// Mitsubishi GX Works2 project: PLC_250924최종   PLC: Q03UDE

// global labels: Global1
VAR_GLOBAL
  H속도변경 AT D10 : INT;
  H축1현재위치 AT D100 : DINT;
  H축2현재위치 AT D104 : DINT;
  H축1에러번호 AT D110 : INT;
  H축2에러번호 AT D111 : INT;
  H축1경고번호 AT D112 : INT;
  H축2경고번호 AT D113 : INT;
  H축1위치1 AT D120 : DINT;
  H축2위치2 AT D140 : DINT;
  H조그속도값 AT D160 : INT;
  H축1기동번호 AT D200 : DINT;
  축2기동 AT M1 : BOOL;
  H시작 AT M10 : BOOL;
  H속도변경버튼 AT M13 : BOOL;
  H축1위치1입력 AT M101 : BOOL;
  H축1위치2입력 AT M102 : BOOL;
  H축1위치3입력 AT M103 : BOOL;
  H축2위치1입력 AT M105 : BOOL;
  H축2위치2입력 AT M106 : BOOL;
  H축1위치1기동명령 AT M111 : BOOL;
  H축1위치2기동명령 AT M112 : BOOL;
  H축1위치3기동명령 AT M113 : BOOL;
  H축2위치1기동명령 AT M115 : BOOL;
  H축2위치2기동명령 AT M116 : BOOL;
  H조그상 AT M121 : BOOL;
  H조그하 AT M122 : BOOL;
  H조그좌 AT M123 : BOOL;
  H조그우 AT M124 : BOOL;
  H축1원점복귀 AT M125 : BOOL;
  H축2원점복귀 AT M126 : BOOL;
  H롬저장 AT M128 : BOOL;
  H축1서보정지 AT M129 : BOOL;
  H축2서보정지 AT M130 : BOOL;
  H축1기동스위치 AT M200 : BOOL;
  H축2기동스위치 AT M201 : BOOL;
  축1서보기동번호 AT U4\G1500 : INT;
  축2서보기동번호 AT U4\G1600 : INT;
  축1서보에러리셋 AT U4\G1502 : INT;
  축2서보에러리셋 AT U4\G1602 : INT;
  축1조그스피드값 AT U4\G1518 : DINT;
  축2조그스피드값 AT U4\G1618 : DINT;
  서보롬쓰기 AT U4\G1900 : INT;
  축2서보현재위치 AT U4\G900 : DINT;
  축1서보이송속도 AT U4\G804 : DINT;
  축2서보이송속도 AT U4\G904 : DINT;
  축1서보에러번호 AT U4\G806 : INT;
  H축1위치2 AT D124 : DINT;
  H축1위치3 AT D128 : DINT;
  H정지 AT M11 : BOOL;
  H일시정지 AT M12 : BOOL;
  축2서보에러번호 AT U4\G906 : INT;
  축1서보경고번호 AT U4\G807 : INT;
  축2서보경고번호 AT U4\G907 : INT;
  축1원점복귀완료 AT U4\G817.4 : BOOL;
  축2원점복귀완료 AT U4\G917.4 : BOOL;
  QD75레디 AT X40 : BOOL;
  축1서보비지 AT X4C : BOOL;
  축2서보비지 AT X4D : BOOL;
  축1서보완료 AT X54 : BOOL;
  축2서보완료 AT X55 : BOOL;
  PLC레디 AT Y40 : BOOL;
  축1서보정지 AT Y44 : BOOL;
  축2서보정지 AT Y45 : BOOL;
  축1조그정기동 AT Y48 : BOOL;
  축1조그역기동 AT Y49 : BOOL;
  H축2위치1 AT D136 : DINT;
  축2조그정기동 AT Y4A : BOOL;
  H축2기동번호 AT D204 : DINT;
  축2조그역기동 AT Y4B : BOOL;
  축1서보기동 AT Y50 : BOOL;
  축2서보기동 AT Y51 : BOOL;
END_VAR
VAR_GLOBAL CONSTANT
  기계원점복귀 : INT := K9001;
END_VAR
VAR_GLOBAL
  축1서보현재위치 AT U4\G800 : DINT;
  축1기동 AT M0 : BOOL;
  in색판별완료 AT M601 : BOOL;
  in두봇완료 AT M602 : BOOL;
  in흰색게이트오픈 AT M603 : BOOL;
  in검은색게이트오픈 AT M604 : BOOL;
  in흰박스full AT M605 : BOOL;
  in검은박스full AT M606 : BOOL;
  in흰박스AMR적재완 AT M607 : BOOL;
  in검은박스AMR적재완 AT M608 : BOOL;
  out공정시작 AT M700 : BOOL;
  out색판정위치도착 AT M701 : BOOL;
  out바퀴분류위치도착 AT M702 : BOOL;
  out흰박스준비완 AT M703 : BOOL;
  out검은박스준비완 AT M704 : BOOL;
  out서보흰컨베이어도착 AT M705 : BOOL;
  out서보검은컨베이어도착 AT M706 : BOOL;
  out흰박스AMR안착 AT M707 : BOOL;
  out검은박스AMR안착 AT M708 : BOOL;
  바퀴매거진센서 AT X0 : BOOL;
  바퀴공급전진센서 AT X1 : BOOL;
  바퀴공급후진센서 AT X2 : BOOL;
  바퀴차단전진센서 AT X3 : BOOL;
  바퀴차단후진센서 AT X4 : BOOL;
  바퀴판정위치센서 AT X5 : BOOL;
  바퀴분류위치센서 AT X6 : BOOL;
  흰박스매거진센서 AT X9 : BOOL;
  흰박스공급후진센서 AT X0A : BOOL;
  흰박스공급전진센서 AT X0B : BOOL;
  흰박스차단위치센서 AT X0C : BOOL;
  흰박스도착위치센서 AT X0D : BOOL;
  검은박스매거진센서 AT X0E : BOOL;
  검은박스공급전진센서 AT X0F : BOOL;
  검은박스공급후진센서 AT X10 : BOOL;
  검은박스차단위치센서 AT X11 : BOOL;
  검은박스도착위치센서 AT X12 : BOOL;
  그리퍼전진센서 AT X15 : BOOL;
  그리퍼후진센서 AT X16 : BOOL;
  그리퍼CW센서 AT X13 : BOOL;
  그리퍼CCW센서 AT X14 : BOOL;
  H축2위치3 AT D144 : DINT;
  H축2위치3입력 AT M107 : BOOL;
  H축2위치3기동명령 AT M117 : BOOL;
  H축2위치4 AT D148 : DINT;
  H축1위치4 AT D132 : DINT;
  H축1위치4입력 AT M104 : BOOL;
  H축2위치4입력 AT M108 : BOOL;
  H축1위치4기동명령 AT M114 : BOOL;
  H축2위치4기동명령 AT M118 : BOOL;
  H에러리셋 AT M127 : BOOL;
  H축2위치5 AT D152 : DINT;
  H축2위치5입력 AT M109 : BOOL;
  H축2위치5기동명령 AT M119 : BOOL;
  비상정지버튼 AT X17 : BOOL;
  바퀴공급전진솔 AT Y20 : BOOL;
  바퀴공급후진솔 AT Y21 : BOOL;
  바퀴차단전진솔 AT Y22 : BOOL;
  바퀴차단후진솔 AT Y23 : BOOL;
  바퀴컨베이어모터구동 AT Y24 : BOOL;
  흰박스공급전진솔 AT Y25 : BOOL;
  흰박스공급후진솔 AT Y26 : BOOL;
  흰박스컨베이어모터구동 AT Y27 : BOOL;
  검은박스공급전진솔 AT Y28 : BOOL;
  검은박스공급후진솔 AT Y29 : BOOL;
  검은박스컨베이어모터구동 AT Y2A : BOOL;
  그리퍼전진솔 AT Y2B : BOOL;
  그리퍼후진솔 AT Y2C : BOOL;
  그리퍼CW솔 AT Y2D : BOOL;
  그리퍼CCW솔 AT Y2E : BOOL;
  경광녹색 AT Y2F : BOOL;
  경광황색 AT Y30 : BOOL;
  경광적색 AT Y31 : BOOL;
  H전체공정시작신호 AT M500 : BOOL;
  H수동조작모드 AT M501 : BOOL;
  H바퀴공급전후진 AT M502 : BOOL;
  H바퀴차단전후진 AT M503 : BOOL;
  H바퀴컨베이어 AT M504 : BOOL;
  H흰박스공급전후진 AT M505 : BOOL;
  H흰박스컨베이어 AT M506 : BOOL;
  H검은박스공급전후진 AT M507 : BOOL;
  H검은박스컨베이어 AT M508 : BOOL;
  H그리퍼전후진 AT M509 : BOOL;
  H그리퍼각도12 AT M510 : BOOL;
  H실린더리셋 AT M511 : BOOL;
  H흰바퀴수 AT D1000 : INT;
  H검은바퀴수 AT D1001 : INT;
  H불량바퀴수 AT D1002 : INT;
  H흰박스수 AT D1003 : INT;
  H검은박스수 AT D1004 : INT;
  OUT신호리셋 AT M1000 : BOOL;
  in공정리셋 AT M609 : BOOL;
  in흰바퀴 AT M610 : BOOL;
  in검은바퀴 AT M611 : BOOL;
  in파란바퀴 AT M612 : BOOL;
END_VAR

PROGRAM MAIN
VAR
  흰박스시작 : BOOL;
  흰박스컨베이어구동 : BOOL;
  흰박스공급전진 : BOOL;
  흰박스공급후진 : BOOL;
  T흰박스차단도착 : TIMER;
  흰박스공정완료 : BOOL;
  검은박스시작 : BOOL;
  검은박스컨베이어구동 : BOOL;
  곰운박스공급전진 : BOOL;
  검은박스공급전진 : BOOL;
  검은박스공급후진 : BOOL;
  T검은박스차단도착 : TIMER;
  검은박스공정완료 : BOOL;
  바퀴공정시작 : BOOL;
  바퀴컨베이어구동 : BOOL;
  바퀴공급전진 : BOOL;
  바퀴차단전진 : BOOL;
  바퀴공급후진 : BOOL;
  T바퀴컨베이어일시정지 : TIMER;
  바퀴컨베이어재구동 : BOOL;
  바퀴공정종료 : BOOL;
  바취차단후진 : BOOL;
  바퀴차단후진 : BOOL;
  T바퀴분류위치도착 : TIMER;
  서보이동시작 : BOOL;
  그리퍼CW : BOOL;
  그리퍼CCW : BOOL;
  흰컨위치이동 : BOOL;
  흰박스컨베이어재구동 : BOOL;
  T흰박스도착위치 : TIMER;
  검은컨위치이동 : BOOL;
  검은박스컨베이어재구동 : BOOL;
  T검은박스도착위치 : TIMER;
  그리퍼전진 : BOOL;
  흰컨업위치이동 : BOOL;
  AMR적재위치이동 : BOOL;
  AMR푸시위치이동 : BOOL;
  푸시 : BOOL;
  원점이동 : BOOL;
  원점복귀 : BOOL;
  흰박스이송완료 : BOOL;
  검은컨업위치이동 : BOOL;
  검은박스이송완료 : BOOL;
  그리퍼후진 : BOOL;
  AMR푸시준비 : BOOL;
  AMR푸쉬준비 : BOOL;
  AMR적재완료 : BOOL;
  축1흰컨위치이동 : BOOL;
  축2흰컨위치이동 : BOOL;
  축2흰컨위치동 : BOOL;
  축1검은컨위치이동 : BOOL;
  축2검은컨위치이동 : BOOL;
  AMR축1적재위치이동 : BOOL;
  AMR축2적재위치이동 : BOOL;
  AMR축1푸시준비 : BOOL;
  AMR축2푸시준비 : BOOL;
  T바퀴매거진없음 : TIMER;
  그리퍼CW1 : BOOL;
  그리퍼CCW1 : BOOL;
  그리퍼전진1 : BOOL;
  그리퍼후진1 : BOOL;
  그리퍼CW2 : BOOL;
  그리퍼CCW2 : BOOL;
  그리퍼전진2 : BOOL;
  그리퍼후진2 : BOOL;
  그리퍼CCW0 : BOOL;
  그리퍼후진0 : BOOL;
  그리퍼ccw0컷 : BOOL;
  그리퍼후진0컷 : BOOL;
  검은박스위치 : BOOL;
  흰박스위치 : BOOL;
  공정중 : BOOL;
  공정종료 : BOOL;
  파란불 : BOOL;
  노란불 : BOOL;
  빨간불1 : BOOL;
  빨간불2 : BOOL;
  빨간불 : BOOL;
  리셋바퀴공급후진 : BOOL;
  리셋바퀴차단후진 : BOOL;
  리셋흰박스공급후진 : BOOL;
  리셋검은박스공급후진 : BOOL;
  리셋그리퍼후진 : BOOL;
  리셋그리퍼CCW : BOOL;
  cut리셋바퀴공급후진 : BOOL;
  cut리셋바퀴차단후진 : BOOL;
  cut리셋흰박스공급후진 : BOOL;
  cut리셋검은박스공급후진 : BOOL;
  cut리셋그리퍼후진 : BOOL;
  cut리셋그리퍼CCW : BOOL;
  T흰박스매거진없음 : TIMER;
  T검은박스매거진없음 : TIMER;
  흰박스진행중 : BOOL;
  검은박스진행중 : BOOL;
  축1원점복귀 : BOOL;
  축2원점복귀 : BOOL;
  흰바퀴수 : INT;
  검은바퀴수 : INT;
  불량바퀴수 : INT;
  흰박스수 : INT;
  검은박스수 : INT;
  노란불파란불끊기용 : BOOL;
END_VAR
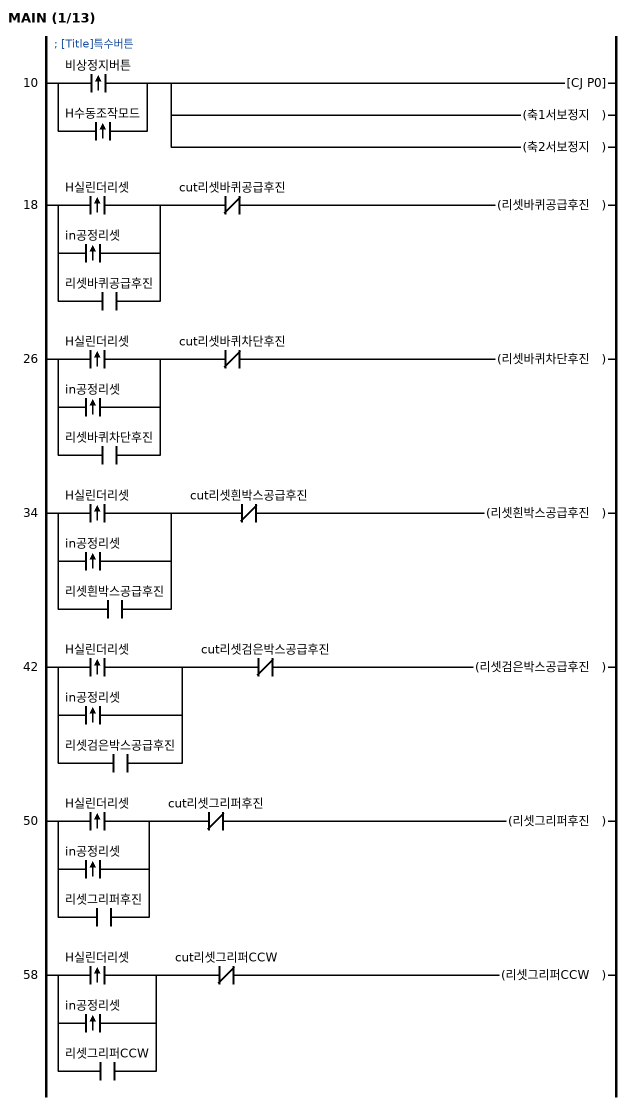
; [Title]특수버튼
10    LDP     비상정지버튼
      ORP     H수동조작모드
      CJ      P0
      OUT     축1서보정지
      OUT     축2서보정지
18    LDP     H실린더리셋
      ORP     in공정리셋
      OR      리셋바퀴공급후진
      ANI     cut리셋바퀴공급후진
      OUT     리셋바퀴공급후진
26    LDP     H실린더리셋
      ORP     in공정리셋
      OR      리셋바퀴차단후진
      ANI     cut리셋바퀴차단후진
      OUT     리셋바퀴차단후진
34    LDP     H실린더리셋
      ORP     in공정리셋
      OR      리셋흰박스공급후진
      ANI     cut리셋흰박스공급후진
      OUT     리셋흰박스공급후진
42    LDP     H실린더리셋
      ORP     in공정리셋
      OR      리셋검은박스공급후진
      ANI     cut리셋검은박스공급후진
      OUT     리셋검은박스공급후진
50    LDP     H실린더리셋
      ORP     in공정리셋
      OR      리셋그리퍼후진
      ANI     cut리셋그리퍼후진
      OUT     리셋그리퍼후진
58    LDP     H실린더리셋
      ORP     in공정리셋
      OR      리셋그리퍼CCW
      ANI     cut리셋그리퍼CCW
      OUT     리셋그리퍼CCW
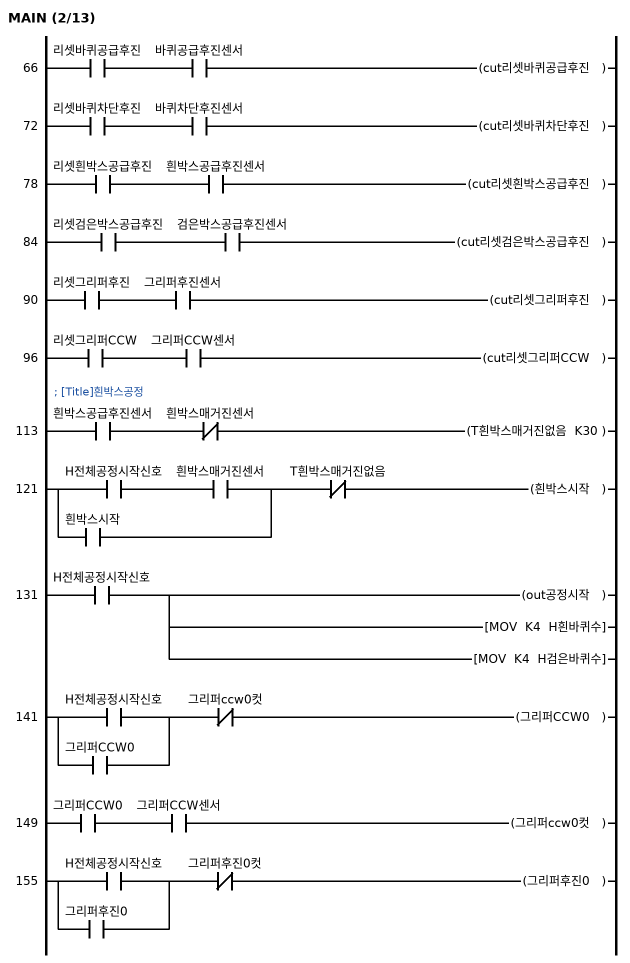
66    LD      리셋바퀴공급후진
      AND     바퀴공급후진센서
      OUT     cut리셋바퀴공급후진
72    LD      리셋바퀴차단후진
      AND     바퀴차단후진센서
      OUT     cut리셋바퀴차단후진
78    LD      리셋흰박스공급후진
      AND     흰박스공급후진센서
      OUT     cut리셋흰박스공급후진
84    LD      리셋검은박스공급후진
      AND     검은박스공급후진센서
      OUT     cut리셋검은박스공급후진
90    LD      리셋그리퍼후진
      AND     그리퍼후진센서
      OUT     cut리셋그리퍼후진
96    LD      리셋그리퍼CCW
      AND     그리퍼CCW센서
      OUT     cut리셋그리퍼CCW
; [Title]흰박스공정
113   LD      흰박스공급후진센서
      ANI     흰박스매거진센서
      OUT     T흰박스매거진없음 K30
121   LD      H전체공정시작신호
      AND     흰박스매거진센서
      OR      흰박스시작
      ANI     T흰박스매거진없음
      OUT     흰박스시작
131   LD      H전체공정시작신호
      OUT     out공정시작
      MOV     K4 H흰바퀴수
      MOV     K4 H검은바퀴수
141   LD      H전체공정시작신호
      OR      그리퍼CCW0
      ANI     그리퍼ccw0컷
      OUT     그리퍼CCW0
149   LD      그리퍼CCW0
      AND     그리퍼CCW센서
      OUT     그리퍼ccw0컷
155   LD      H전체공정시작신호
      OR      그리퍼후진0
      ANI     그리퍼후진0컷
      OUT     그리퍼후진0
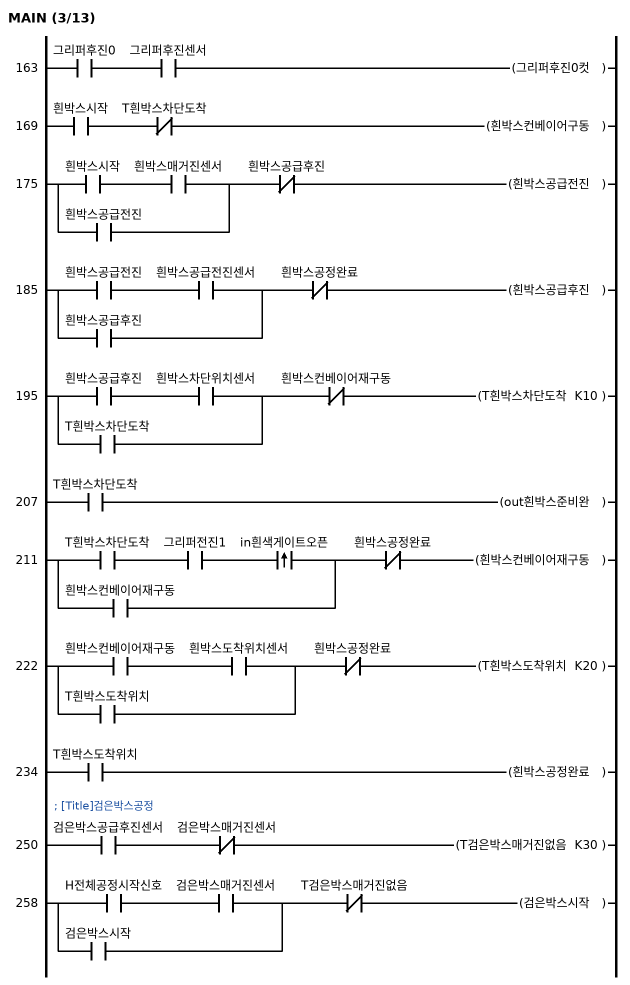
163   LD      그리퍼후진0
      AND     그리퍼후진센서
      OUT     그리퍼후진0컷
169   LD      흰박스시작
      ANI     T흰박스차단도착
      OUT     흰박스컨베이어구동
175   LD      흰박스시작
      AND     흰박스매거진센서
      OR      흰박스공급전진
      ANI     흰박스공급후진
      OUT     흰박스공급전진
185   LD      흰박스공급전진
      AND     흰박스공급전진센서
      OR      흰박스공급후진
      ANI     흰박스공정완료
      OUT     흰박스공급후진
195   LD      흰박스공급후진
      AND     흰박스차단위치센서
      OR      T흰박스차단도착
      ANI     흰박스컨베이어재구동
      OUT     T흰박스차단도착 K10
207   LD      T흰박스차단도착
      OUT     out흰박스준비완
211   LD      T흰박스차단도착
      AND     그리퍼전진1
      ANDP    in흰색게이트오픈
      OR      흰박스컨베이어재구동
      ANI     흰박스공정완료
      OUT     흰박스컨베이어재구동
222   LD      흰박스컨베이어재구동
      AND     흰박스도착위치센서
      OR      T흰박스도착위치
      ANI     흰박스공정완료
      OUT     T흰박스도착위치 K20
234   LD      T흰박스도착위치
      OUT     흰박스공정완료
; [Title]검은박스공정
250   LD      검은박스공급후진센서
      ANI     검은박스매거진센서
      OUT     T검은박스매거진없음 K30
258   LD      H전체공정시작신호
      AND     검은박스매거진센서
      OR      검은박스시작
      ANI     T검은박스매거진없음
      OUT     검은박스시작
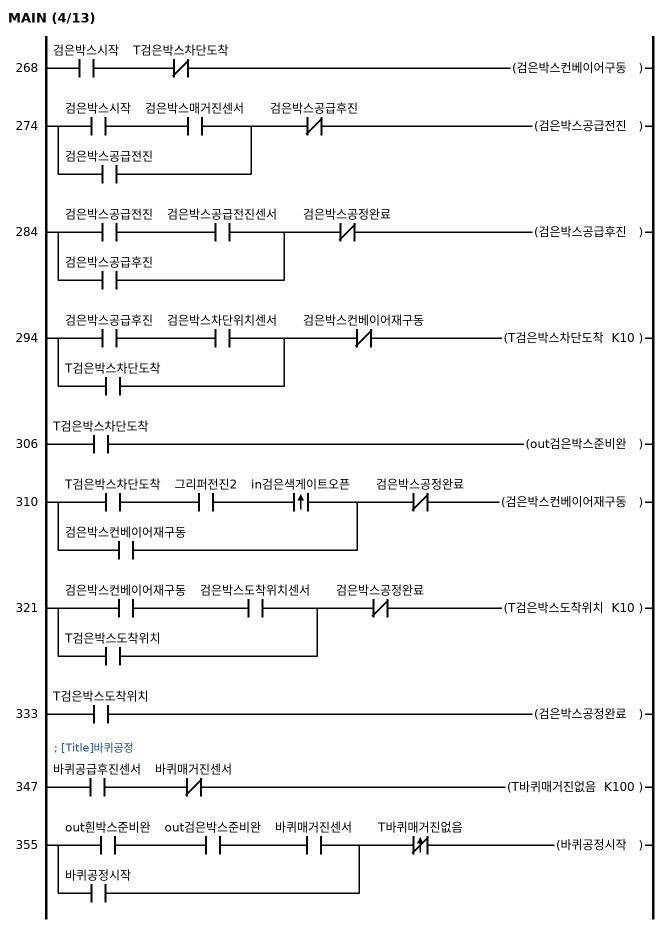
268   LD      검은박스시작
      ANI     T검은박스차단도착
      OUT     검은박스컨베이어구동
274   LD      검은박스시작
      AND     검은박스매거진센서
      OR      검은박스공급전진
      ANI     검은박스공급후진
      OUT     검은박스공급전진
284   LD      검은박스공급전진
      AND     검은박스공급전진센서
      OR      검은박스공급후진
      ANI     검은박스공정완료
      OUT     검은박스공급후진
294   LD      검은박스공급후진
      AND     검은박스차단위치센서
      OR      T검은박스차단도착
      ANI     검은박스컨베이어재구동
      OUT     T검은박스차단도착 K10
306   LD      T검은박스차단도착
      OUT     out검은박스준비완
310   LD      T검은박스차단도착
      AND     그리퍼전진2
      ANDP    in검은색게이트오픈
      OR      검은박스컨베이어재구동
      ANI     검은박스공정완료
      OUT     검은박스컨베이어재구동
321   LD      검은박스컨베이어재구동
      AND     검은박스도착위치센서
      OR      T검은박스도착위치
      ANI     검은박스공정완료
      OUT     T검은박스도착위치 K10
333   LD      T검은박스도착위치
      OUT     검은박스공정완료
; [Title]바퀴공정
347   LD      바퀴공급후진센서
      ANI     바퀴매거진센서
      OUT     T바퀴매거진없음 K100
355   LD      out흰박스준비완
      AND     out검은박스준비완
      AND     바퀴매거진센서
      OR      바퀴공정시작
      ANDPI   T바퀴매거진없음
      OUT     바퀴공정시작
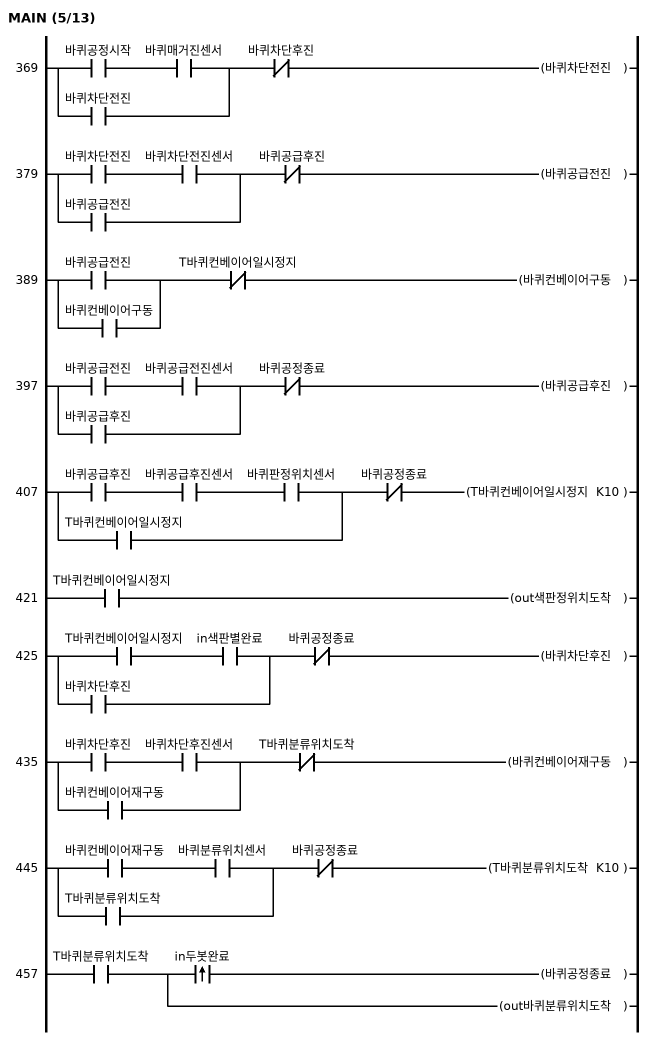
369   LD      바퀴공정시작
      AND     바퀴매거진센서
      OR      바퀴차단전진
      ANI     바퀴차단후진
      OUT     바퀴차단전진
379   LD      바퀴차단전진
      AND     바퀴차단전진센서
      OR      바퀴공급전진
      ANI     바퀴공급후진
      OUT     바퀴공급전진
389   LD      바퀴공급전진
      OR      바퀴컨베이어구동
      ANI     T바퀴컨베이어일시정지
      OUT     바퀴컨베이어구동
397   LD      바퀴공급전진
      AND     바퀴공급전진센서
      OR      바퀴공급후진
      ANI     바퀴공정종료
      OUT     바퀴공급후진
407   LD      바퀴공급후진
      AND     바퀴공급후진센서
      AND     바퀴판정위치센서
      OR      T바퀴컨베이어일시정지
      ANI     바퀴공정종료
      OUT     T바퀴컨베이어일시정지 K10
421   LD      T바퀴컨베이어일시정지
      OUT     out색판정위치도착
425   LD      T바퀴컨베이어일시정지
      AND     in색판별완료
      OR      바퀴차단후진
      ANI     바퀴공정종료
      OUT     바퀴차단후진
435   LD      바퀴차단후진
      AND     바퀴차단후진센서
      OR      바퀴컨베이어재구동
      ANI     T바퀴분류위치도착
      OUT     바퀴컨베이어재구동
445   LD      바퀴컨베이어재구동
      AND     바퀴분류위치센서
      OR      T바퀴분류위치도착
      ANI     바퀴공정종료
      OUT     T바퀴분류위치도착 K10
457   LD      T바퀴분류위치도착
      MPS
      ANDP    in두봇완료
      OUT     바퀴공정종료
      MPP
      OUT     out바퀴분류위치도착
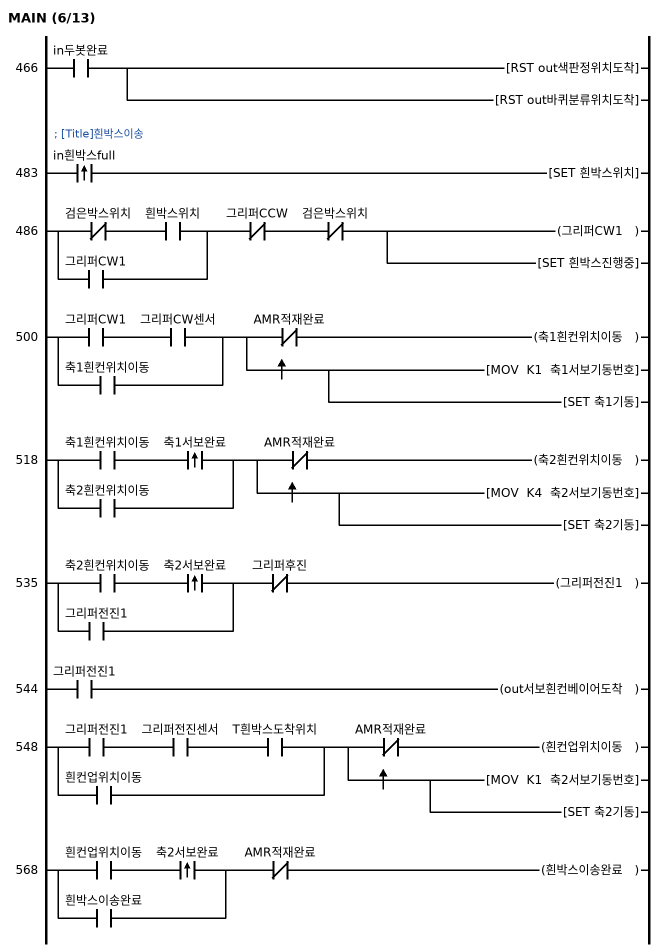
466   LD      in두봇완료
      RST     out색판정위치도착
      RST     out바퀴분류위치도착
; [Title]흰박스이송
483   LDP     in흰박스full
      SET     흰박스위치
486   LDI     검은박스위치
      AND     흰박스위치
      OR      그리퍼CW1
      ANI     그리퍼CCW
      ANI     검은박스위치
      OUT     그리퍼CW1
      SET     흰박스진행중
500   LD      그리퍼CW1
      AND     그리퍼CW센서
      OR      축1흰컨위치이동
      MPS
      ANI     AMR적재완료
      OUT     축1흰컨위치이동
      MPP
      MEP
      MOV     K1 축1서보기동번호
      SET     축1기동
518   LD      축1흰컨위치이동
      ANDP    축1서보완료
      OR      축2흰컨위치이동
      MPS
      ANI     AMR적재완료
      OUT     축2흰컨위치이동
      MPP
      MEP
      MOV     K4 축2서보기동번호
      SET     축2기동
535   LD      축2흰컨위치이동
      ANDP    축2서보완료
      OR      그리퍼전진1
      ANI     그리퍼후진
      OUT     그리퍼전진1
544   LD      그리퍼전진1
      OUT     out서보흰컨베이어도착
548   LD      그리퍼전진1
      AND     그리퍼전진센서
      AND     T흰박스도착위치
      OR      흰컨업위치이동
      MPS
      ANI     AMR적재완료
      OUT     흰컨업위치이동
      MPP
      MEP
      MOV     K1 축2서보기동번호
      SET     축2기동
568   LD      흰컨업위치이동
      ANDP    축2서보완료
      OR      흰박스이송완료
      ANI     AMR적재완료
      OUT     흰박스이송완료
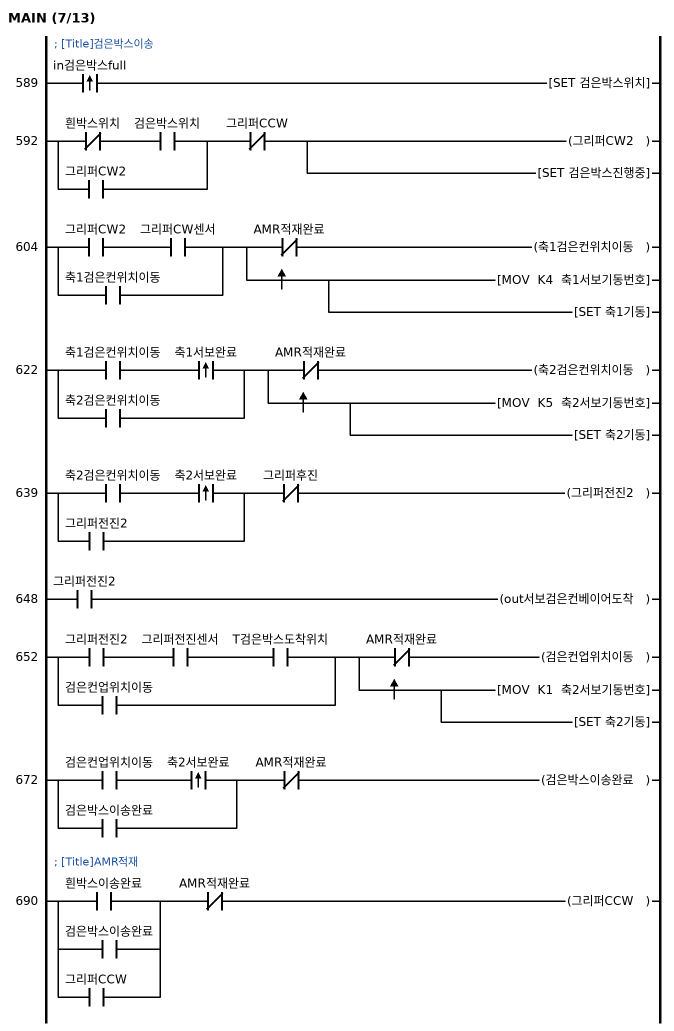
; [Title]검은박스이송
589   LDP     in검은박스full
      SET     검은박스위치
592   LDI     흰박스위치
      AND     검은박스위치
      OR      그리퍼CW2
      ANI     그리퍼CCW
      OUT     그리퍼CW2
      SET     검은박스진행중
604   LD      그리퍼CW2
      AND     그리퍼CW센서
      OR      축1검은컨위치이동
      MPS
      ANI     AMR적재완료
      OUT     축1검은컨위치이동
      MPP
      MEP
      MOV     K4 축1서보기동번호
      SET     축1기동
622   LD      축1검은컨위치이동
      ANDP    축1서보완료
      OR      축2검은컨위치이동
      MPS
      ANI     AMR적재완료
      OUT     축2검은컨위치이동
      MPP
      MEP
      MOV     K5 축2서보기동번호
      SET     축2기동
639   LD      축2검은컨위치이동
      ANDP    축2서보완료
      OR      그리퍼전진2
      ANI     그리퍼후진
      OUT     그리퍼전진2
648   LD      그리퍼전진2
      OUT     out서보검은컨베이어도착
652   LD      그리퍼전진2
      AND     그리퍼전진센서
      AND     T검은박스도착위치
      OR      검은컨업위치이동
      MPS
      ANI     AMR적재완료
      OUT     검은컨업위치이동
      MPP
      MEP
      MOV     K1 축2서보기동번호
      SET     축2기동
672   LD      검은컨업위치이동
      ANDP    축2서보완료
      OR      검은박스이송완료
      ANI     AMR적재완료
      OUT     검은박스이송완료
; [Title]AMR적재
690   LD      흰박스이송완료
      OR      검은박스이송완료
      OR      그리퍼CCW
      ANI     AMR적재완료
      OUT     그리퍼CCW
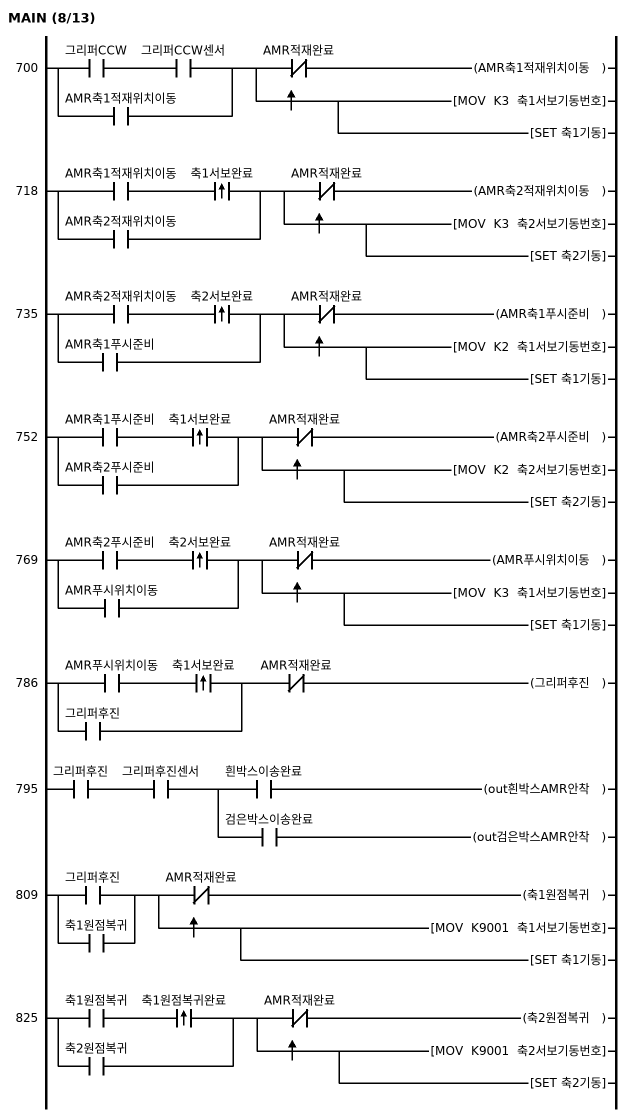
700   LD      그리퍼CCW
      AND     그리퍼CCW센서
      OR      AMR축1적재위치이동
      MPS
      ANI     AMR적재완료
      OUT     AMR축1적재위치이동
      MPP
      MEP
      MOV     K3 축1서보기동번호
      SET     축1기동
718   LD      AMR축1적재위치이동
      ANDP    축1서보완료
      OR      AMR축2적재위치이동
      MPS
      ANI     AMR적재완료
      OUT     AMR축2적재위치이동
      MPP
      MEP
      MOV     K3 축2서보기동번호
      SET     축2기동
735   LD      AMR축2적재위치이동
      ANDP    축2서보완료
      OR      AMR축1푸시준비
      MPS
      ANI     AMR적재완료
      OUT     AMR축1푸시준비
      MPP
      MEP
      MOV     K2 축1서보기동번호
      SET     축1기동
752   LD      AMR축1푸시준비
      ANDP    축1서보완료
      OR      AMR축2푸시준비
      MPS
      ANI     AMR적재완료
      OUT     AMR축2푸시준비
      MPP
      MEP
      MOV     K2 축2서보기동번호
      SET     축2기동
769   LD      AMR축2푸시준비
      ANDP    축2서보완료
      OR      AMR푸시위치이동
      MPS
      ANI     AMR적재완료
      OUT     AMR푸시위치이동
      MPP
      MEP
      MOV     K3 축1서보기동번호
      SET     축1기동
786   LD      AMR푸시위치이동
      ANDP    축1서보완료
      OR      그리퍼후진
      ANI     AMR적재완료
      OUT     그리퍼후진
795   LD      그리퍼후진
      AND     그리퍼후진센서
      MPS
      AND     흰박스이송완료
      OUT     out흰박스AMR안착
      MPP
      AND     검은박스이송완료
      OUT     out검은박스AMR안착
809   LD      그리퍼후진
      OR      축1원점복귀
      MPS
      ANI     AMR적재완료
      OUT     축1원점복귀
      MPP
      MEP
      MOV     K9001 축1서보기동번호
      SET     축1기동
825   LD      축1원점복귀
      ANDP    축1원점복귀완료
      OR      축2원점복귀
      MPS
      ANI     AMR적재완료
      OUT     축2원점복귀
      MPP
      MEP
      MOV     K9001 축2서보기동번호
      SET     축2기동
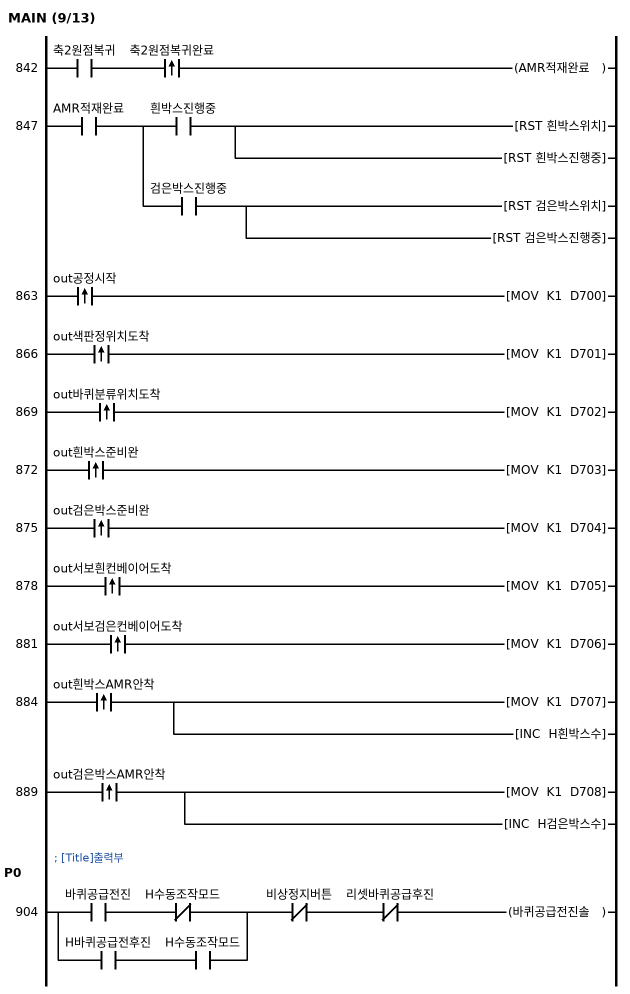
842   LD      축2원점복귀
      ANDP    축2원점복귀완료
      OUT     AMR적재완료
847   LD      AMR적재완료
      MPS
      AND     흰박스진행중
      RST     흰박스위치
      RST     흰박스진행중
      MPP
      AND     검은박스진행중
      RST     검은박스위치
      RST     검은박스진행중
863   LDP     out공정시작
      MOV     K1 D700
866   LDP     out색판정위치도착
      MOV     K1 D701
869   LDP     out바퀴분류위치도착
      MOV     K1 D702
872   LDP     out흰박스준비완
      MOV     K1 D703
875   LDP     out검은박스준비완
      MOV     K1 D704
878   LDP     out서보흰컨베이어도착
      MOV     K1 D705
881   LDP     out서보검은컨베이어도착
      MOV     K1 D706
884   LDP     out흰박스AMR안착
      MOV     K1 D707
      INC     H흰박스수
889   LDP     out검은박스AMR안착
      MOV     K1 D708
      INC     H검은박스수
; [Title]출력부
      P0
904   LD      바퀴공급전진
      ANI     H수동조작모드
      LD      H바퀴공급전후진
      AND     H수동조작모드
      ORB
      ANI     비상정지버튼
      ANI     리셋바퀴공급후진
      OUT     바퀴공급전진솔
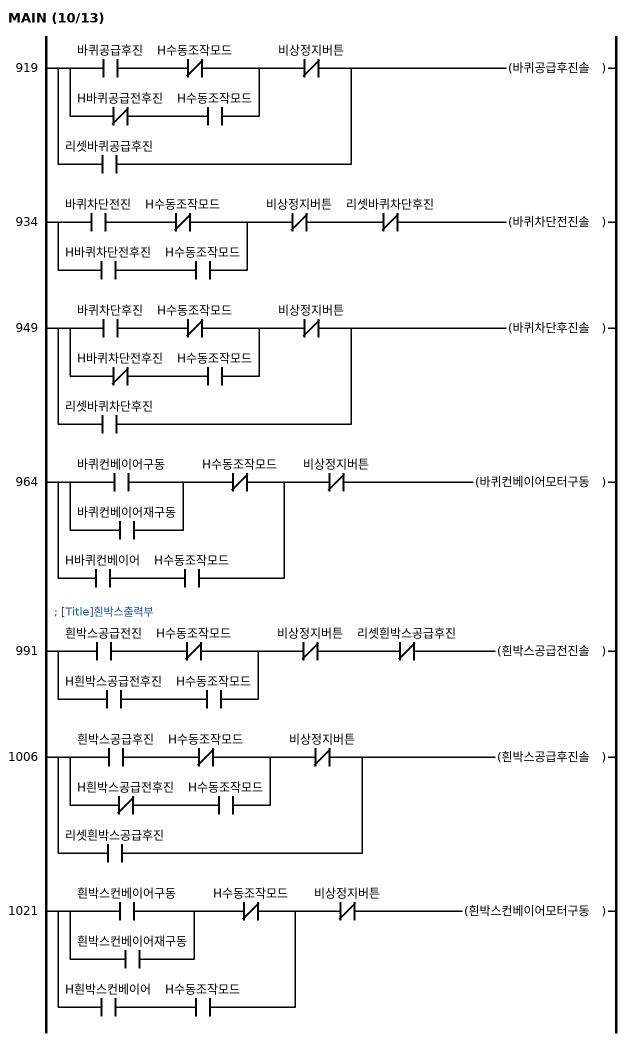
919   LD      바퀴공급후진
      ANI     H수동조작모드
      LDI     H바퀴공급전후진
      AND     H수동조작모드
      ORB
      ANI     비상정지버튼
      OR      리셋바퀴공급후진
      OUT     바퀴공급후진솔
934   LD      바퀴차단전진
      ANI     H수동조작모드
      LD      H바퀴차단전후진
      AND     H수동조작모드
      ORB
      ANI     비상정지버튼
      ANI     리셋바퀴차단후진
      OUT     바퀴차단전진솔
949   LD      바퀴차단후진
      ANI     H수동조작모드
      LDI     H바퀴차단전후진
      AND     H수동조작모드
      ORB
      ANI     비상정지버튼
      OR      리셋바퀴차단후진
      OUT     바퀴차단후진솔
964   LD      바퀴컨베이어구동
      OR      바퀴컨베이어재구동
      ANI     H수동조작모드
      LD      H바퀴컨베이어
      AND     H수동조작모드
      ORB
      ANI     비상정지버튼
      OUT     바퀴컨베이어모터구동
; [Title]흰박스출력부
991   LD      흰박스공급전진
      ANI     H수동조작모드
      LD      H흰박스공급전후진
      AND     H수동조작모드
      ORB
      ANI     비상정지버튼
      ANI     리셋흰박스공급후진
      OUT     흰박스공급전진솔
1006  LD      흰박스공급후진
      ANI     H수동조작모드
      LDI     H흰박스공급전후진
      AND     H수동조작모드
      ORB
      ANI     비상정지버튼
      OR      리셋흰박스공급후진
      OUT     흰박스공급후진솔
1021  LD      흰박스컨베이어구동
      OR      흰박스컨베이어재구동
      ANI     H수동조작모드
      LD      H흰박스컨베이어
      AND     H수동조작모드
      ORB
      ANI     비상정지버튼
      OUT     흰박스컨베이어모터구동
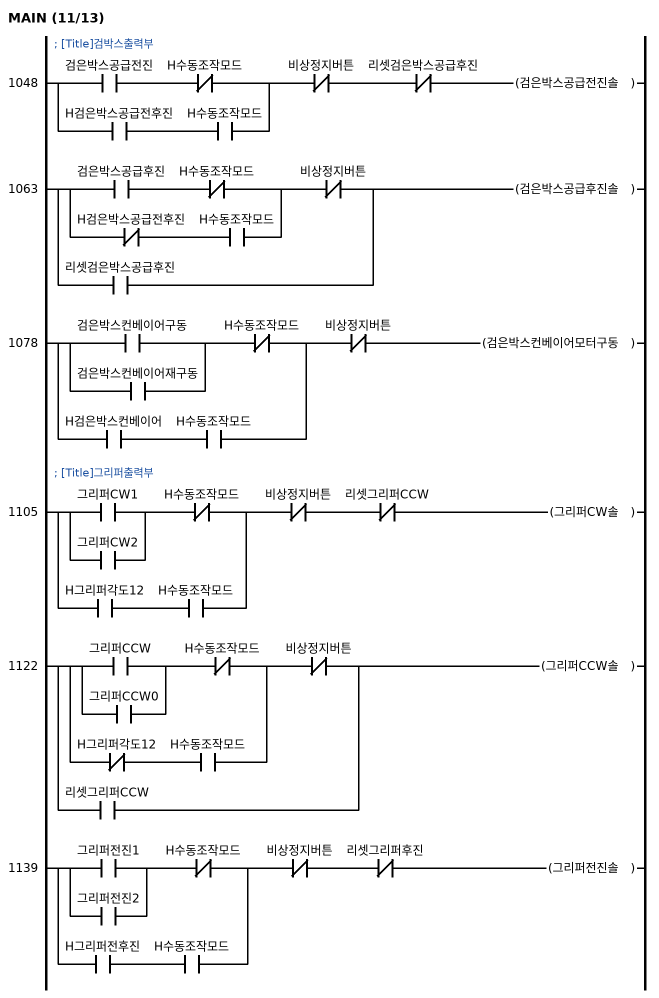
; [Title]검박스출력부
1048  LD      검은박스공급전진
      ANI     H수동조작모드
      LD      H검은박스공급전후진
      AND     H수동조작모드
      ORB
      ANI     비상정지버튼
      ANI     리셋검은박스공급후진
      OUT     검은박스공급전진솔
1063  LD      검은박스공급후진
      ANI     H수동조작모드
      LDI     H검은박스공급전후진
      AND     H수동조작모드
      ORB
      ANI     비상정지버튼
      OR      리셋검은박스공급후진
      OUT     검은박스공급후진솔
1078  LD      검은박스컨베이어구동
      OR      검은박스컨베이어재구동
      ANI     H수동조작모드
      LD      H검은박스컨베이어
      AND     H수동조작모드
      ORB
      ANI     비상정지버튼
      OUT     검은박스컨베이어모터구동
; [Title]그리퍼출력부
1105  LD      그리퍼CW1
      OR      그리퍼CW2
      ANI     H수동조작모드
      LD      H그리퍼각도12
      AND     H수동조작모드
      ORB
      ANI     비상정지버튼
      ANI     리셋그리퍼CCW
      OUT     그리퍼CW솔
1122  LD      그리퍼CCW
      OR      그리퍼CCW0
      ANI     H수동조작모드
      LDI     H그리퍼각도12
      AND     H수동조작모드
      ORB
      ANI     비상정지버튼
      OR      리셋그리퍼CCW
      OUT     그리퍼CCW솔
1139  LD      그리퍼전진1
      OR      그리퍼전진2
      ANI     H수동조작모드
      LD      H그리퍼전후진
      AND     H수동조작모드
      ORB
      ANI     비상정지버튼
      ANI     리셋그리퍼후진
      OUT     그리퍼전진솔
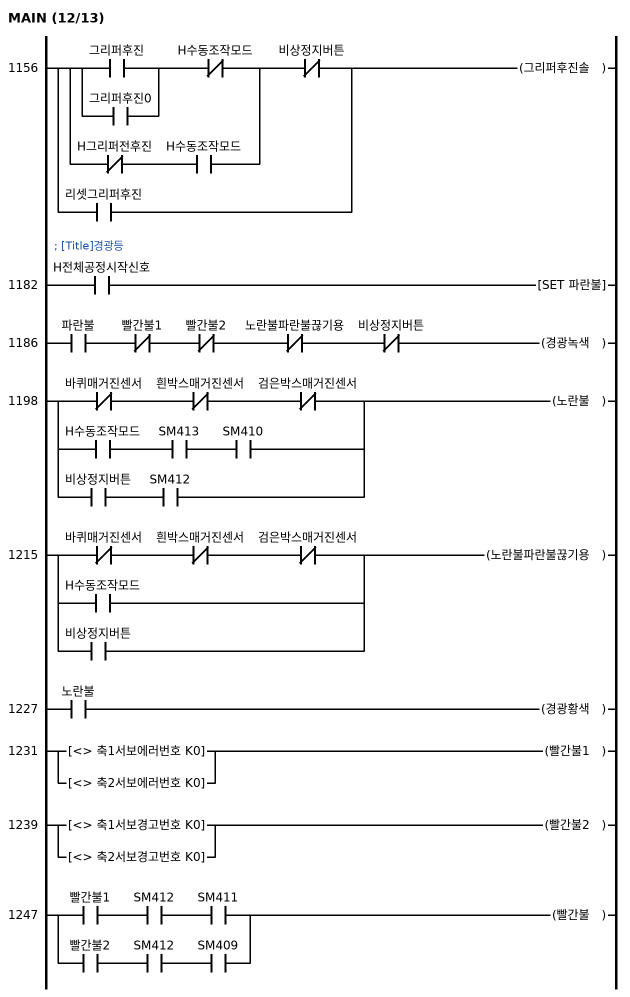
1156  LD      그리퍼후진
      OR      그리퍼후진0
      ANI     H수동조작모드
      LDI     H그리퍼전후진
      AND     H수동조작모드
      ORB
      ANI     비상정지버튼
      OR      리셋그리퍼후진
      OUT     그리퍼후진솔
; [Title]경광등
1182  LD      H전체공정시작신호
      SET     파란불
1186  LD      파란불
      ANI     빨간불1
      ANI     빨간불2
      ANI     노란불파란불끊기용
      ANI     비상정지버튼
      OUT     경광녹색
1198  LDI     바퀴매거진센서
      ANI     흰박스매거진센서
      ANI     검은박스매거진센서
      LD      H수동조작모드
      AND     SM413
      AND     SM410
      ORB
      LD      비상정지버튼
      AND     SM412
      ORB
      OUT     노란불
1215  LDI     바퀴매거진센서
      ANI     흰박스매거진센서
      ANI     검은박스매거진센서
      OR      H수동조작모드
      OR      비상정지버튼
      OUT     노란불파란불끊기용
1227  LD      노란불
      OUT     경광황색
1231  LD<>    축1서보에러번호 K0
      OR<>    축2서보에러번호 K0
      OUT     빨간불1
1239  LD<>    축1서보경고번호 K0
      OR<>    축2서보경고번호 K0
      OUT     빨간불2
1247  LD      빨간불1
      AND     SM412
      AND     SM411
      LD      빨간불2
      AND     SM412
      AND     SM409
      ORB
      OUT     빨간불
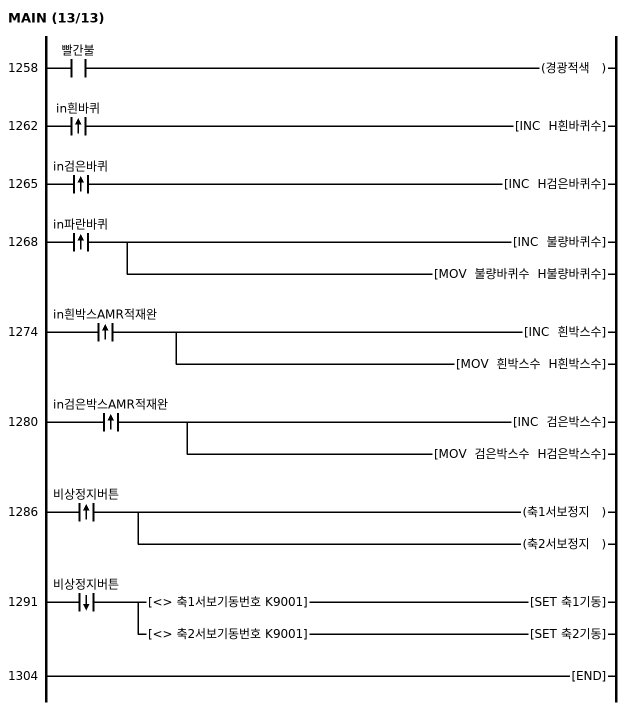
1258  LD      빨간불
      OUT     경광적색
1262  LDP     in흰바퀴
      INC     H흰바퀴수
1265  LDP     in검은바퀴
      INC     H검은바퀴수
1268  LDP     in파란바퀴
      INC     불량바퀴수
      MOV     불량바퀴수 H불량바퀴수
1274  LDP     in흰박스AMR적재완
      INC     흰박스수
      MOV     흰박스수 H흰박스수
1280  LDP     in검은박스AMR적재완
      INC     검은박스수
      MOV     검은박스수 H검은박스수
1286  LDP     비상정지버튼
      OUT     축1서보정지
      OUT     축2서보정지
1291  LDF     비상정지버튼
      MPS
      AND<>   축1서보기동번호 K9001
      SET     축1기동
      MPP
      AND<>   축2서보기동번호 K9001
      SET     축2기동
1304  END
END_PROGRAM

PROGRAM SERVO
VAR
  서보준비완료 : BOOL;
  축1사용자조그속도 : DINT;
  축2사용자조그속도 : DINT;
  서준 : BOOL;
  테스트1 : BOOL;
  테스트2 : BOOL;
END_VAR
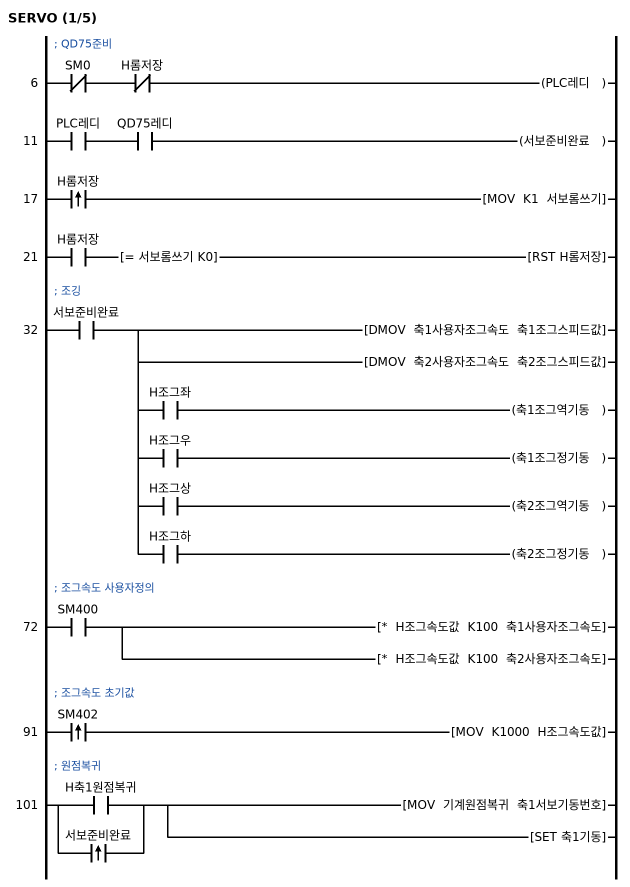
; QD75준비
6     LDI     SM0
      ANI     H롬저장
      OUT     PLC레디
11    LD      PLC레디
      AND     QD75레디
      OUT     서보준비완료
17    LDP     H롬저장
      MOV     K1 서보롬쓰기
21    LD      H롬저장
      AND=    서보롬쓰기 K0
      RST     H롬저장
; 조깅
32    LD      서보준비완료
      DMOV    축1사용자조그속도 축1조그스피드값
      DMOV    축2사용자조그속도 축2조그스피드값
      MPS
      AND     H조그좌
      OUT     축1조그역기동
      MRD
      AND     H조그우
      OUT     축1조그정기동
      MRD
      AND     H조그상
      OUT     축2조그역기동
      MPP
      AND     H조그하
      OUT     축2조그정기동
; 조그속도 사용자정의
72    LD      SM400
      *       H조그속도값 K100 축1사용자조그속도
      *       H조그속도값 K100 축2사용자조그속도
; 조그속도 초기값
91    LDP     SM402
      MOV     K1000 H조그속도값
; 원점복귀
101   LD      H축1원점복귀
      ORP     서보준비완료
      MOV     기계원점복귀 축1서보기동번호
      SET     축1기동
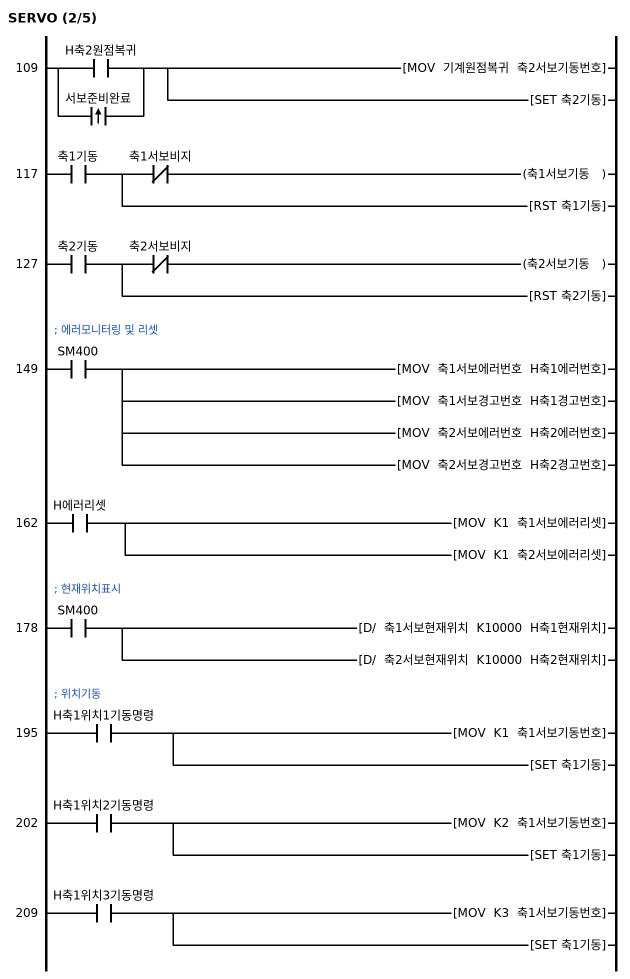
109   LD      H축2원점복귀
      ORP     서보준비완료
      MOV     기계원점복귀 축2서보기동번호
      SET     축2기동
117   LD      축1기동
      MPS
      ANI     축1서보비지
      OUT     축1서보기동
      MPP
      RST     축1기동
127   LD      축2기동
      MPS
      ANI     축2서보비지
      OUT     축2서보기동
      MPP
      RST     축2기동
; 에러모니터링 및 리셋
149   LD      SM400
      MOV     축1서보에러번호 H축1에러번호
      MOV     축1서보경고번호 H축1경고번호
      MOV     축2서보에러번호 H축2에러번호
      MOV     축2서보경고번호 H축2경고번호
162   LD      H에러리셋
      MOV     K1 축1서보에러리셋
      MOV     K1 축2서보에러리셋
; 현재위치표시
178   LD      SM400
      D/      축1서보현재위치 K10000 H축1현재위치
      D/      축2서보현재위치 K10000 H축2현재위치
; 위치기동
195   LD      H축1위치1기동명령
      MOV     K1 축1서보기동번호
      SET     축1기동
202   LD      H축1위치2기동명령
      MOV     K2 축1서보기동번호
      SET     축1기동
209   LD      H축1위치3기동명령
      MOV     K3 축1서보기동번호
      SET     축1기동
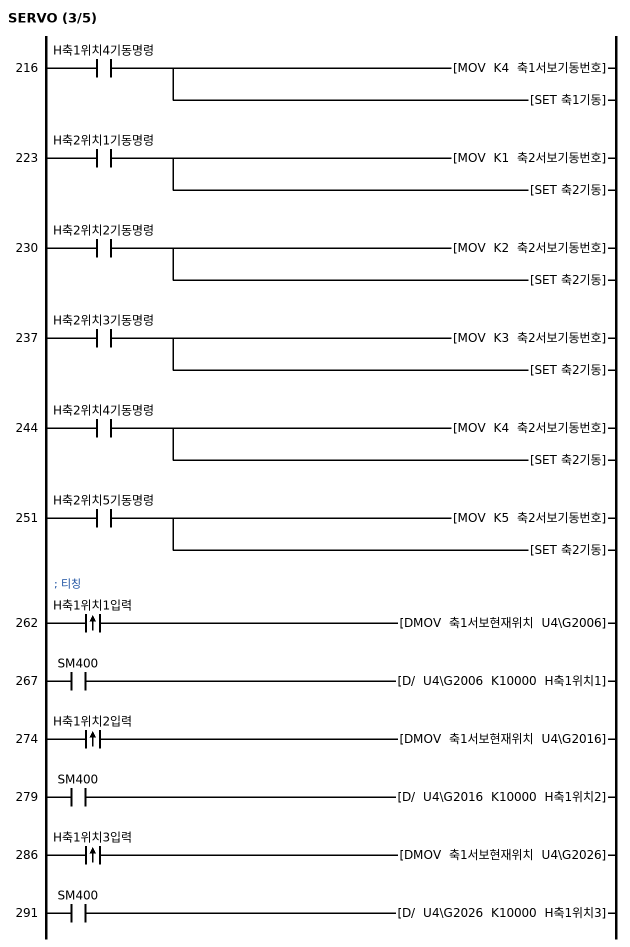
216   LD      H축1위치4기동명령
      MOV     K4 축1서보기동번호
      SET     축1기동
223   LD      H축2위치1기동명령
      MOV     K1 축2서보기동번호
      SET     축2기동
230   LD      H축2위치2기동명령
      MOV     K2 축2서보기동번호
      SET     축2기동
237   LD      H축2위치3기동명령
      MOV     K3 축2서보기동번호
      SET     축2기동
244   LD      H축2위치4기동명령
      MOV     K4 축2서보기동번호
      SET     축2기동
251   LD      H축2위치5기동명령
      MOV     K5 축2서보기동번호
      SET     축2기동
; 티칭
262   LDP     H축1위치1입력
      DMOV    축1서보현재위치 U4\G2006
267   LD      SM400
      D/      U4\G2006 K10000 H축1위치1
274   LDP     H축1위치2입력
      DMOV    축1서보현재위치 U4\G2016
279   LD      SM400
      D/      U4\G2016 K10000 H축1위치2
286   LDP     H축1위치3입력
      DMOV    축1서보현재위치 U4\G2026
291   LD      SM400
      D/      U4\G2026 K10000 H축1위치3
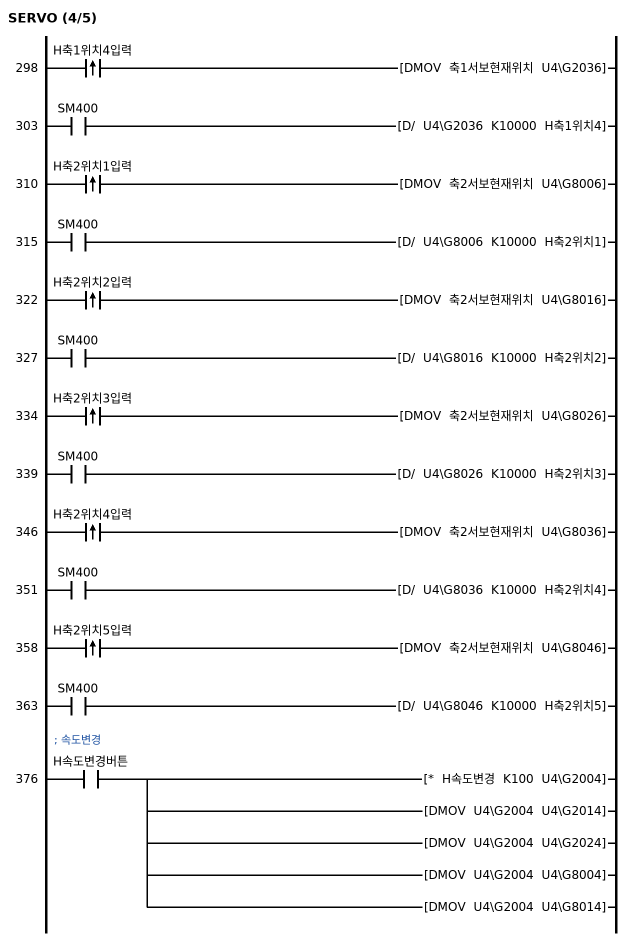
298   LDP     H축1위치4입력
      DMOV    축1서보현재위치 U4\G2036
303   LD      SM400
      D/      U4\G2036 K10000 H축1위치4
310   LDP     H축2위치1입력
      DMOV    축2서보현재위치 U4\G8006
315   LD      SM400
      D/      U4\G8006 K10000 H축2위치1
322   LDP     H축2위치2입력
      DMOV    축2서보현재위치 U4\G8016
327   LD      SM400
      D/      U4\G8016 K10000 H축2위치2
334   LDP     H축2위치3입력
      DMOV    축2서보현재위치 U4\G8026
339   LD      SM400
      D/      U4\G8026 K10000 H축2위치3
346   LDP     H축2위치4입력
      DMOV    축2서보현재위치 U4\G8036
351   LD      SM400
      D/      U4\G8036 K10000 H축2위치4
358   LDP     H축2위치5입력
      DMOV    축2서보현재위치 U4\G8046
363   LD      SM400
      D/      U4\G8046 K10000 H축2위치5
; 속도변경
376   LD      H속도변경버튼
      *       H속도변경 K100 U4\G2004
      DMOV    U4\G2004 U4\G2014
      DMOV    U4\G2004 U4\G2024
      DMOV    U4\G2004 U4\G8004
      DMOV    U4\G2004 U4\G8014
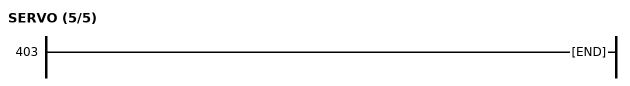
403   END
END_PROGRAM
